Omron CX-Programmer project NewProject (CX-Programmer 9.51)

# PLC my_first_project: CP1L L
; comment

## Program NewProgram1 (cyclic task 0)
Local symbols
button_1 0.00 BOOL  ; comment
button_2 0.01 BOOL  ; comment
button_3 0.02 BOOL  ; comment
out_2 100.01 BOOL  ; comment

### Section Section1

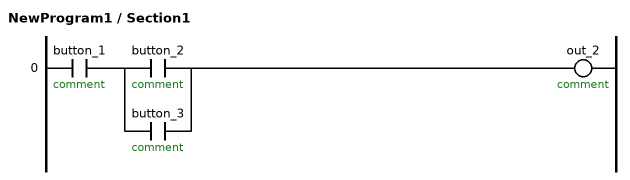
; rung 0
LD button_1  ; comment
LD button_2  ; comment
OR button_3  ; comment
ANDLD
OUT out_2  ; comment

### Section END
; rung 0
END(001)